// Mitsubishi GX Works2 project: Conveyor safety   PLC: FX1N/FX1NC

PROGRAM MAIN
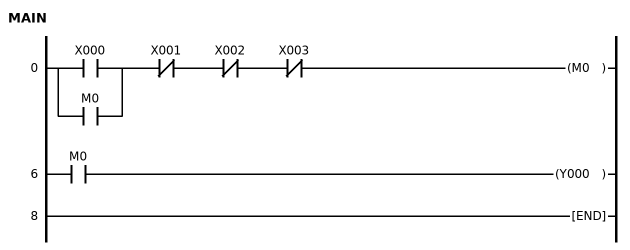
0     LD      X000
      OR      M0
      ANI     X001
      ANI     X002
      ANI     X003
      OUT     M0
6     LD      M0
      OUT     Y000
8     END
END_PROGRAM
